FUNCTION_BLOCK FB_BIN_MANAGER
VAR_INPUT
	Enable	: BOOL;
END_VAR
VAR_OUTPUT
	FrontForkValve	: FB_HYDRAULIC_VALVE;
	RearForkValve	: FB_HYDRAULIC_VALVE;
	GateStop		: BOOL;
	Error			: BOOL;
	Ready			: BOOL;
END_VAR
VAR
	State 		: (DEFAULT, INIT, IDLE, LOAD, UNLOAD, ERROR);
	PrevState	: (DEFAULT, INIT, IDLE, LOAD, UNLOAD, ERROR);
	StateEntry	: BOOL;
END_VAR



IF State <> PrevState THEN
	StateEntry := TRUE;
	PrevState := State;
ELSE
	StateEntry := FALSE;
END_IF

CASE State OF
	DEFAULT:
		//
	INIT:
		//
	IDLE:
		//
	LOAD:
		//
	UNLOAD:
		//
	ERROR:
		//
END_CASE

END_FUNCTION_BLOCK

(* stored: Version 1.1.0.1, ProductVersion 3.1.4024.12
   POU FB_BIN_MANAGER: Id {40c5c23c-1578-445e-b6b1-2a2174ba3b30}, SpecialFunc None *)
